TYPE ST_ManualSection EXTENDS ST_SectionBase :
STRUCT
	nAutoMan		: UINT; //0 manual, 1 auto
	nManForward		: UINT;
	nManBackward	: UINT;
	nManLeft		: UINT;
	nManRight		: UINT;
	fManDriveSpeed	: REAL;
END_STRUCT
END_TYPE

(* stored: Version 1.1.0.1, ProductVersion 3.1.4024.12
   DUT ST_ManualSection: Id {867cd426-fbf2-40b5-a692-3cf6763d0ba8} *)
